SUBAPPLICATION GreenWhiteBackground (* Subapplication Type *)
  (* Standard: 61499-2 *)
  (* Version 1.0, 2022-11-10, franz *)
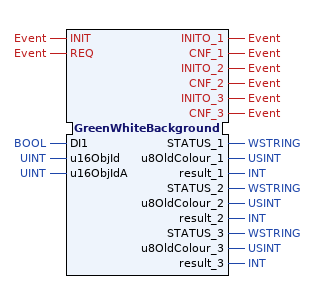
  EVENT_INPUT
    INIT; (* Initialization Request *)
    REQ; (* Normal Execution Request *)
  END_EVENT
  EVENT_OUTPUT
    INITO_1; (* Initialization Confirm *)
    CNF_1; (* Execution Confirmation *)
    INITO_2;
    CNF_2;
    INITO_3;
    CNF_3;
  END_EVENT
  VAR_INPUT
    DI1 : BOOL; (* Selector *)
    u16ObjId : UINT; (* Object ID Softkey *)
    u16ObjIdA : UINT; (* Object ID AUX *)
  END_VAR
  VAR_OUTPUT
    STATUS_1 : WSTRING; (* Service Status *)
    u8OldColour_1 : USINT; (* Old value of ID *)
    result_1 : INT; (* retval see description *)
    STATUS_2 : WSTRING; (* Service Status *)
    u8OldColour_2 : USINT; (* Old value of ID *)
    result_2 : INT; (* retval see description *)
    STATUS_3 : WSTRING; (* Service Status *)
    u8OldColour_3 : USINT; (* Old value of ID *)
    result_3 : INT; (* retval see description *)
  END_VAR
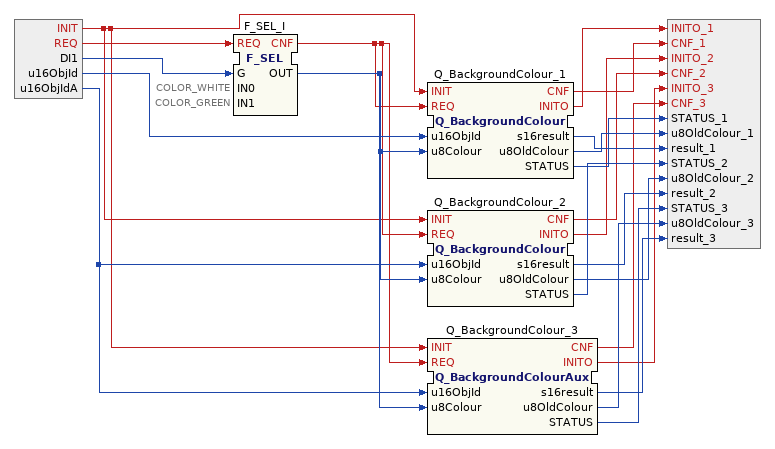
  FBS
    Q_BackgroundColour_1 : Q_BackgroundColour;
    Q_BackgroundColour_2 : Q_BackgroundColour;
    Q_BackgroundColour_3 : Q_BackgroundColourAux;
    F_SEL_I : F_SEL(IN0 := COLOR_WHITE, IN1 := COLOR_GREEN);
  END_FBS
  EVENT_CONNECTIONS
    INIT TO Q_BackgroundColour_1.INIT;
    INIT TO Q_BackgroundColour_2.INIT;
    INIT TO Q_BackgroundColour_3.INIT;
    Q_BackgroundColour_3.CNF TO CNF_3;
    Q_BackgroundColour_2.CNF TO CNF_2;
    Q_BackgroundColour_1.CNF TO CNF_1;
    Q_BackgroundColour_3.INITO TO INITO_3;
    Q_BackgroundColour_2.INITO TO INITO_2;
    Q_BackgroundColour_1.INITO TO INITO_1;
    F_SEL_I.CNF TO Q_BackgroundColour_1.REQ;
    F_SEL_I.CNF TO Q_BackgroundColour_2.REQ;
    F_SEL_I.CNF TO Q_BackgroundColour_3.REQ;
    REQ TO F_SEL_I.REQ;
  END_CONNECTIONS
  DATA_CONNECTIONS
    u16ObjId TO Q_BackgroundColour_1.u16ObjId;
    u16ObjIdA TO Q_BackgroundColour_2.u16ObjId;
    u16ObjIdA TO Q_BackgroundColour_3.u16ObjId;
    Q_BackgroundColour_3.s16result TO result_3;
    Q_BackgroundColour_3.u8OldColour TO u8OldColour_3;
    Q_BackgroundColour_3.STATUS TO STATUS_3;
    Q_BackgroundColour_2.s16result TO result_2;
    Q_BackgroundColour_2.u8OldColour TO u8OldColour_2;
    Q_BackgroundColour_2.STATUS TO STATUS_2;
    Q_BackgroundColour_1.s16result TO result_1;
    Q_BackgroundColour_1.u8OldColour TO u8OldColour_1;
    Q_BackgroundColour_1.STATUS TO STATUS_1;
    F_SEL_I.OUT TO Q_BackgroundColour_1.u8Colour;
    F_SEL_I.OUT TO Q_BackgroundColour_2.u8Colour;
    F_SEL_I.OUT TO Q_BackgroundColour_3.u8Colour;
    DI1 TO F_SEL_I.G;
  END_CONNECTIONS
END_SUBAPPLICATION
